PROGRAM MAIN
VAR
END_VAR


DomParser();
OperatorOverloading_Test();
DynamicArrays_Test();

END_PROGRAM

(* stored: Version 1.1.0.1, ProductVersion 3.1.4024.12
   POU MAIN: Id {05c9249a-2d2a-4719-9e1d-3233a5c387bc}, SpecialFunc None *)
